PROGRAM MAIN
VAR
	velocityX AT%Q* : LREAL;
	velocityY AT%Q* : LREAL;
	theta AT%Q* : LREAL;
END_VAR

velocityX := vars.fromMatlab_velocityX;
velocityY := vars.fromMatlab_velocityY;
theta := vars.fromMatlab_theta;

END_PROGRAM

(* stored: Version 1.1.0.1, ProductVersion 3.1.4022.3
   POU MAIN: Id {7ab232d5-bf67-4c8a-bfe1-11ef0fe8c457}, SpecialFunc None *)
